FUNCTION daysInMonth : INT
VAR_INPUT
	nYear	: INT;
	nMonth	: INT;
END_VAR
VAR
END_VAR

CASE nMonth OF 
	1:
		daysInMonth := 31;
	2:
		daysInMonth := 28 + BOOL_TO_INT(isLeapYear(nYear:= nYear));
	3:
		daysInMonth := 31;
	4:
		daysInMonth := 30;
	5:
		daysInMonth := 31;
	6:
		daysInMonth := 30;
	7:
		daysInMonth := 31;
	8:
		daysInMonth := 31;
	9:
		daysInMonth := 30;
	10:
		daysInMonth := 31;
	11:
		daysInMonth := 30;
	12:
		daysInMonth := 31;
END_CASE

END_FUNCTION

(* stored: Version 1.1.0.1, ProductVersion 3.1.4024.11
   POU daysInMonth: Id {2fd857d9-b017-4cc8-ba65-24cdf21d1743}, SpecialFunc None *)
